(* CODESYS project FU_sPaddFrontBIBO.xml

Project tree, tasks and I/O mapping:
  function FU_sPaddFrontBIBO [ST]
*)

// FU_sPaddFrontBIBO
//This function padds the front of a string with the given character, the given amount
//If the padd amount plus the string is longer than the output string, the input string will be cut off to make space for the padding
// +-----------+----------+----------+-----------------------------------------------------------------------------------------------------------------------+
// |**Version**|**Author**| **Date** |**Changes**                                                                                                            |
// +-----------+----------+----------+-----------------------------------------------------------------------------------------------------------------------+
// | 1         | NSN      | 04-02-19 | Creation                                                                                                              |
// +-----------+----------+----------+-----------------------------------------------------------------------------------------------------------------------+
FUNCTION FU_sPaddFrontBIBO : BOOL
VAR_IN_OUT
	sOut		:STRING(1);			//Output String
	sStr		:STRING(1);			//Input String
END_VAR
VAR_INPUT
	wPadds		:WORD;				//How much to padd it
	wOutSize	:WORD;				//Output String Size
	eChar		:EASCII;		//Which character to padd with
END_VAR
VAR
	In1Add		:POINTER TO BYTE;	//Address of first string
	StrAdd		:POINTER TO BYTE;	//Address of output string
END_VAR

In1Add					:=		ADR(sStr);
StrAdd					:=		ADR(sOut);
IF wPadds = 0 THEN
	WHILE wOutSize > 0 DO
		wOutSize		:=		wOutSize - 1;
		IF In1Add^ <> 0 THEN
			StrAdd^		:=		In1Add^;
			In1Add		:=		In1Add + 1;
		ELSE
			EXIT;
		END_IF
		StrAdd			:=		StrAdd + 1;
	END_WHILE
	StrAdd^				:=		EASCII.Null;
ELSE
	WHILE wOutSize > 0 DO
		wOutSize		:=		wOutSize - 1;
		IF wPadds > 0 THEN
			StrAdd^		:=		eChar;
			wPadds		:=		wPadds - 1;
		ELSIF In1Add^ <> 0 THEN
			StrAdd^		:=		In1Add^;
			In1Add		:=		In1Add + 1;
		ELSE
			EXIT;
		END_IF
		StrAdd			:=		StrAdd + 1;
	END_WHILE
	StrAdd^				:=		EASCII.Null;
END_IF

END_FUNCTION
